% RSLogix 500 project project3.RSS, saved by version 8.30.00.16 %
PROJECT "UNTITLED"    % processor: Bul.1763 MicroLogix 1100 Series B %

PROGRAM FILES
  LAD 2 "MAIN"  9 rungs

DATA FILES
  O0 OUTPUT  4 elements
  I1 INPUT  6 elements
  S2 STATUS  66 elements
  B3 BINARY  2 elements
  T4 TIMER  1 elements
  C5 COUNTER  1 elements
  R6 CONTROL  1 elements
  N7 INTEGER  4 elements
  F8 FLOAT  1 elements
  ST9 STRING  10 elements

LADDER 2 "MAIN"
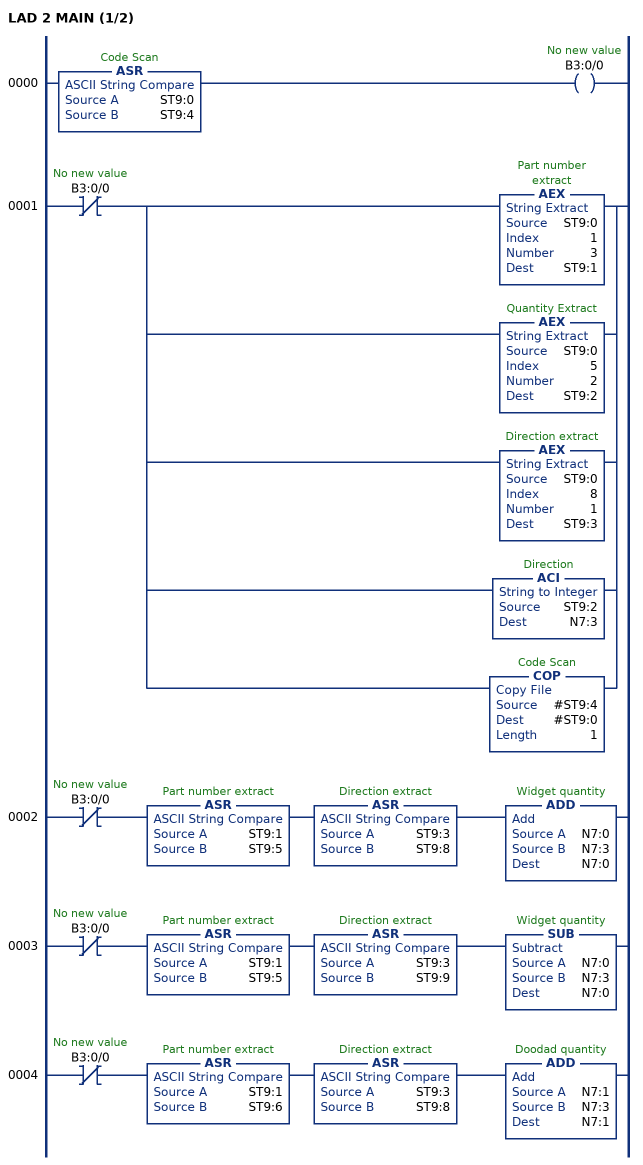
% Rung: 0 %
SOR ASR ST9:0 ST9:4 OTE B3:0/0 EOR
%   ST9:0  "Code Scan" %
%   ST9:4  "Null string" %
%   B3:0/0  "No new value" %
% Rung: 1 %
SOR XIO B3:0/0 BST AEX ST9:0 1 3 ST9:1 NXB AEX ST9:0 5 2 ST9:2 NXB AEX ST9:0 8 1 ST9:3 NXB ACI ST9:2 N7:3 NXB COP #ST9:4 #ST9:0 1 BND EOR
%   B3:0/0  "No new value" %
%   ST9:0  "Code Scan" %
%   ST9:1  "Part number extract" %
%   ST9:2  "Quantity Extract" %
%   ST9:3  "Direction extract" %
%   N7:3  "Direction" %
%   ST9:4  "Null string" %
% Rung: 2 %
SOR XIO B3:0/0 ASR ST9:1 ST9:5 ASR ST9:3 ST9:8 ADD N7:0 N7:3 N7:0 EOR
%   B3:0/0  "No new value" %
%   ST9:1  "Part number extract" %
%   ST9:5  "123 compare" %
%   ST9:3  "Direction extract" %
%   ST9:8  "Incoming dir" %
%   N7:0  "Widget quantity" %
%   N7:3  "Direction" %
% Rung: 3 %
SOR XIO B3:0/0 ASR ST9:1 ST9:5 ASR ST9:3 ST9:9 SUB N7:0 N7:3 N7:0 EOR
%   B3:0/0  "No new value" %
%   ST9:1  "Part number extract" %
%   ST9:5  "123 compare" %
%   ST9:3  "Direction extract" %
%   ST9:9  "Outgoing dir" %
%   N7:0  "Widget quantity" %
%   N7:3  "Direction" %
% Rung: 4 %
SOR XIO B3:0/0 ASR ST9:1 ST9:6 ASR ST9:3 ST9:8 ADD N7:1 N7:3 N7:1 EOR
%   B3:0/0  "No new value" %
%   ST9:1  "Part number extract" %
%   ST9:6  "456 compare" %
%   ST9:3  "Direction extract" %
%   ST9:8  "Incoming dir" %
%   N7:1  "Doodad quantity" %
%   N7:3  "Direction" %

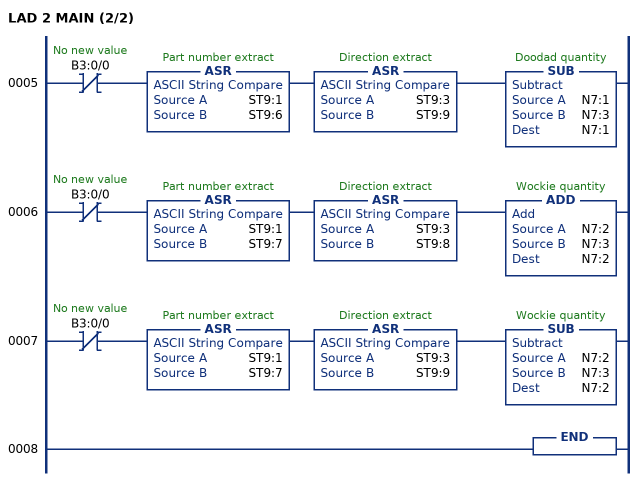
% Rung: 5 %
SOR XIO B3:0/0 ASR ST9:1 ST9:6 ASR ST9:3 ST9:9 SUB N7:1 N7:3 N7:1 EOR
%   B3:0/0  "No new value" %
%   ST9:1  "Part number extract" %
%   ST9:6  "456 compare" %
%   ST9:3  "Direction extract" %
%   ST9:9  "Outgoing dir" %
%   N7:1  "Doodad quantity" %
%   N7:3  "Direction" %
% Rung: 6 %
SOR XIO B3:0/0 ASR ST9:1 ST9:7 ASR ST9:3 ST9:8 ADD N7:2 N7:3 N7:2 EOR
%   B3:0/0  "No new value" %
%   ST9:1  "Part number extract" %
%   ST9:7  "789 compare" %
%   ASR ST9:7  "Direction check" %
%   ST9:3  "Direction extract" %
%   ST9:8  "Incoming dir" %
%   N7:2  "Wockie quantity" %
%   N7:3  "Direction" %
% Rung: 7 %
SOR XIO B3:0/0 ASR ST9:1 ST9:7 ASR ST9:3 ST9:9 SUB N7:2 N7:3 N7:2 EOR
%   B3:0/0  "No new value" %
%   ST9:1  "Part number extract" %
%   ST9:7  "789 compare" %
%   ASR ST9:7  "Direction check" %
%   ST9:3  "Direction extract" %
%   ST9:9  "Outgoing dir" %
%   N7:2  "Wockie quantity" %
%   N7:3  "Direction" %
% Rung: 8 %
SOR END EOR

OTHER DOCUMENTED ADDRESSES
  B3:0/1  "ONS"
  B3:0/2  "String S/E Trigger"
  B3:0/3  "String Reset"
  B3:0/4  "ONS"
  B3:0/5  "String Reset Trigger"
  B3:0/6  "Direction trigger"
  B3:0/7  "Direction Trigger"
  B3:0/8  "ONS"
  B3:0/9  "ONS"
  B3:0/11  "ONS"
  B3:0/12  "ONS"
  B3:1/0  "trigger"

OTHER INSTRUCTION COMMENTS
  ST9:1 ACI  "Conversion"

DATA TABLE (non-zero values as saved)
DATA ST9
% ST9:5 % "123"
% ST9:6 % "456"
% ST9:7 % "789"
% ST9:8 % "1"
% ST9:9 % "2"
